# EPICS substitutions: apps/caenHvApp/Db/seq/ahdcOnOff.substitutions
file "db/ahdcOnOff.db" {
pattern { ONOFF VAL }
        { OFF   0   }
        { ON    1   }
}
